{attribute 'qualified_only'}
VAR_GLOBAL
	//Zmienne obslugi bledow
	bError										: BOOL;														// Zmienna ogolna wystapienia bledu                                                                         							
	udiErrorID									: UDINT;													// Kod bledu 	
	sErrorDescription1							: STRING(200);												// Opis bledu 1
	sErrorDescription2							: STRING(200);												// Opis bledu 2
	sStationInError								: STRING(200);												// Nazwa stacji w bledzie
                                                 
                                                                        	

	tonResettingTime							: TON;														// Licznik odliczacy czas wykonywania procedury resetu
	
	iStep										: INT;														// Krok proedury czytania bledow 	

END_VAR


VAR_GLOBAL CONSTANT
	iErrorStructuresNumber						: INT					:= 9;								// Liczba strukur bledow stacji  w tym strukura bledow globalnych
END_VAR

(* stored: Version 1.1.0.1, FileIdentifier 0737679291abe7f953aa4449a62f1991847a5757, FileSignature 15cff35c5590527cf58e7e384bb385d5fad928ff37364dee4c5ab2088d7a78d7bb8933552c85c361e40a1068b1ce7c1acee19affc38c4a0abba7db04ce0ae62a533f43b4caf1fed177178ac66b90141a209f5caec1434b7670073a820d326ff462f7c5643712b7374853c39f26bdaf6ba598ebdff2a5fdb752527d0b5d259de28f96cf1c0c6b9ef0c682bd4b31ca579c5f61c91d279b2bebebd8669de3739806f4c0b2af4fbbbb1f1f8aad4ce75c61294677bafef6b0a1ef499562f095375870f378dc43afbc09715c9f1a6289ef4ff6f95df6578c8dc07902bc7f8991afb10d02c46f8496e6fe6d6a82d3f04b690de9eb9b2118aeef23956267e42790458cd5
   GVL GVL_ErrorHandling: Id {f8cee543-ed9f-48bc-8fb2-eb267339ca07} *)
